FUNCTION_BLOCK SignalTower
VAR
	lightGreen	: Relay;
	lightRed	: Relay;
END_VAR

PROPERTY GreenLightState : BOOL
GET
GreenLightState := lightGreen.State;
END_GET
END_PROPERTY

PROPERTY RedLightState : BOOL
GET
RedLightState := lightRed.State;
END_GET
END_PROPERTY

METHOD SwitchOffGreen : BOOL
VAR_INPUT
END_VAR
lightGreen.SwitchOff();
END_METHOD

METHOD SwitchOffRed : BOOL
VAR_INPUT
END_VAR
lightRed.SwitchOff();
END_METHOD

METHOD SwitchOnGreen : BOOL
VAR_INPUT
END_VAR
lightGreen.SwitchOn();
END_METHOD

METHOD SwitchOnRed : BOOL
VAR_INPUT
END_VAR
lightRed.SwitchOn();
END_METHOD

END_FUNCTION_BLOCK

(* stored: Version 1.1.0.1
   POU SignalTower: Id {a49b9225-0cc8-4d5e-bdae-213ddc81bbc9}, SpecialFunc None
   Property GreenLightState: Id {f1a7e554-94b8-4cda-8e4c-9796f7d2cf80}
   Get Get: Id {b7bb1740-9fe1-482f-b384-16034c8643b7}
   Property RedLightState: Id {a263101a-c590-4d5a-b8fc-385a84e625e0}
   Get Get: Id {3993bef8-ffef-4e3a-8d3a-704df8851182}
   Method SwitchOffGreen: Id {0b6544a2-3c56-4468-a238-1826e6f830e8}
   Method SwitchOffRed: Id {e965210f-3d87-48d6-869c-5f759f4e9602}
   Method SwitchOnGreen: Id {b3dd5ded-19cc-4e26-8f25-83a7797197f5}
   Method SwitchOnRed: Id {46b231c6-54b4-4b38-84a7-5c86fe779ab4} *)
